// TIA Portal V17 export
// export: Created 2022-07-28T18:03:17.8732362Z, ExportSetting None, DisplayName Totally Integrated Automation Portal, DisplayVersion V17, DisplayName TIA Portal Openness, DisplayVersion V17, DisplayName TIA Portal Teamcenter Gateway, DisplayVersion V17, DisplayName TIA Portal Version Control Interface, DisplayVersion V17, DisplayName TIA Portal Test Suite Advanced, DisplayVersion V17, DisplayName SINAMICS Startdrive Advanced, DisplayVersion V17, DisplayName SINAMICS DCC, DisplayVersion V17, DisplayName SINAMICS Startdrive G130, G150, S120, S150, SINAMICS MV, S210, DisplayVersion V17, DisplayName SINAMICS Startdrive G110M, G120, G120C, G120D, G120P, G115D, DisplayVersion V17, DisplayName STEP 7 Professional, DisplayVersion V17, DisplayName SIMATIC Energy Suite, DisplayVersion V17, DisplayName STEP 7 CFC, DisplayVersion V17, DisplayName STEP 7 Safety, DisplayVersion V17, DisplayName WinCC Advanced / Unified PC, DisplayVersion V17, DisplayName SIMATIC Visualization Architect, DisplayVersion V17
TYPE "Lib_UDT_AutoControl"
   STRUCT
      CLSID : Int := -1;   // Type of element under current index
      Global_CMD { ExternalAccessible := 'False'; ExternalVisible := 'False'; ExternalWritable := 'False'} : Int;   // Command word for element from auto module
      Mode { ExternalAccessible := 'False'; ExternalVisible := 'False'; ExternalWritable := 'False'} : "UDT_Mode";
      StatusGen { ExternalAccessible := 'False'; ExternalVisible := 'False'; ExternalWritable := 'False'} : "_AutoControl_ElementSTW";
      CTW { ExternalAccessible := 'False'; ExternalVisible := 'False'; ExternalWritable := 'False'} : DWord := DWORD#2#0000_0000_0000_0000_0000_0000_0000_0000;   // Control technologie word for control current element
      STW { ExternalAccessible := 'False'; ExternalVisible := 'False'; ExternalWritable := 'False'} : DWord := DWORD#2#0000_0000_0000_0000_0000_0000_0000_0000;   // Status technologie word for control current element
      STW_HMI : DWord;   // Status program word for send data to HMI
      SP_AutoMode { ExternalAccessible := 'False'; ExternalVisible := 'False'; ExternalWritable := 'False'} : Real;   // Setpoint speed/position ... in Auto mode
   END_STRUCT;
END_TYPE
